PROGRAM MACHINE
VAR
END_VAR

IF fbFEEDER.eSTATE= E_STATE.error OR fbSEPARATE1.eSTATE= E_STATE.error THEN
	iMAIN_STATE:=99 ;
END_IF

IF bMAIN_RESET THEN
	iMAIN_STATE:=98 ;
	bMAIN_PAUSE:=FALSE;
	sMAIN_STATE:='UNINIT';
END_IF

CASE iMAIN_STATE OF 
	1: //feeder
		eMAIN_STATE:=E_STATE.busy;
		sMAIN_STATE:='FEEDING';
		fbFEEDER.aSTART();
		IF fbFEEDER.eSTATE= E_STATE.busy THEN
			iMAIN_STATE:=2;
		END_IF
	2://wait for feeder
		IF fbFEEDER.eSTATE= E_STATE.ready THEN
			IF NOT bMAIN_PAUSE THEN
				iMAIN_STATE:=3;
			END_IF
		END_IF
		IF fbFEEDER.eSTATE= E_STATE.error THEN
			iMAIN_STATE:=99;
		END_IF
	3: //separate1
		eMAIN_STATE:=E_STATE.busy;
		sMAIN_STATE:=' SEPARATE1';
		fbSEPARATE1.aSTART();
		IF fbSEPARATE1.eSTATE= E_STATE.busy THEN
			iMAIN_STATE:=4;
		END_IF
	4://wait for separate1
		IF fbSEPARATE1.eSTATE= E_STATE.ready THEN
			IF NOT bMAIN_PAUSE THEN
				iMAIN_STATE:=100;
			END_IF
		END_IF
		IF fbSEPARATE1.eSTATE= E_STATE.error THEN
			iMAIN_STATE:=99;
		END_IF
	98:
		eMAIN_STATE:=E_STATE.uninit;
		sMAIN_STATE:='UNINIT';
		bMAIN_RESET:=FALSE;
		fbFEEDER.aRESET();
		fbSEPARATE1.aRESET();
		//fbPIST3.aRESET();
		IF fbFEEDER.eSTATE = E_STATE.uninit AND fbSEPARATE1.eSTATE = E_STATE.uninit THEN
			iMAIN_STATE:=980;
		END_IF
	980: 
		IF fbFEEDER.eSTATE= E_STATE.ready AND fbSEPARATE1.eSTATE= E_STATE.ready  THEN
			iMAIN_STATE:=100;
		END_IF
		
		IF fbFEEDER.bERROR OR fbSEPARATE1.bERROR THEN
			iMAIN_STATE:=99;
		END_IF
	
	99:
		eMAIN_STATE:=E_STATE.error;
		sMAIN_STATE:='MACHINE ERROR';
		
	100:
		eMAIN_STATE:=E_STATE.ready;
		sMAIN_STATE:='READY';
		IF bMAIN_START THEN
			bMAIN_START:=FALSE;
			iMAIN_STATE:=1;
		END_IF
		
END_CASE

END_PROGRAM

(* stored: Version 1.1.0.1, ProductVersion 3.1.4024.12
   POU MACHINE: Id {9f31af90-0ebb-4c9c-9f88-fd85631a41cf}, SpecialFunc None *)
